// TIA Portal project "项目1" (V16)

(* hardware
DEVICE "HMI_1"  TP1200 Comfort
   slot 0: "HMI_1"  TP1200 Comfort  6AV2 124-0MC01-0AX0  16.0.0.0
   slot 1: "HMI_RT_1"  TP1200 Comfort  6AV2 124-0MC01-0AX0  16.0.0.0
   slot 5: "HMI_1.IE_CP_1"  PROFINET Interface  16.0.0.0
      slot 1: "PROFINET Interface_1"  PROFINET Interface
         slot 1: "Port_1"  Port
         slot 2: "Port_2"  Port
   slot 7: "HMI_1.MPI/DP_CP_1"  MPI/DP Interface  16.0.0.0
DEVICE "S7-1200 station_1"  S7-1200 Station
   slot 0: "Rack_0"  S7-1200 Rack  Rack  V1.0
   slot 1: "PLC_1"  CPU 1214C DC/DC/DC  6ES7 214-1AG40-0XB0  V4.4
*)

// ===== PLC "PLC_1"  CPU 1214C DC/DC/DC =====

VAR_GLOBAL   // PLC tag table "默认变量表"
   "正向" AT %M2.0 : Bool;
   "正向转动" AT %Q0.0 : Bool;
   "反向" AT %M2.1 : Bool;
   "停止" AT %M2.2 : Bool;
   "反向转动" AT %Q0.1 : Bool;
   "Clock_Byte" AT %MB100 : Byte;
   "Clock_10Hz" AT %M100.0 : Bool;
   "Clock_5Hz" AT %M100.1 : Bool;
   "Clock_2Hz" AT %M100.3 : Bool;
   "Clock_1.25Hz" AT %M100.4 : Bool;
   "Clock_1Hz" AT %M100.5 : Bool;   // 已用
   "Clock_0.625Hz" AT %M100.6 : Bool;
   "Clock_0.5Hz" AT %M100.7 : Bool;   // 已用
   "tag1" AT %M0.0 : Bool;
   "tag2" AT %M0.1 : Bool;
   "tag3" AT %M100.2 : Bool;   // 已用
   "tag4" AT %MW10 : Word;
   "tag6" AT %M1.3 : Bool;
   "低水位" AT %M3.0 : Bool;
   "高水位" AT %M3.2 : Bool;
   "供水泵" AT %M3.3 : Bool;
   "抽水" AT %M3.4 : Bool;
   "抽水泵" AT %M3.5 : Bool;
   "箭头动画2" AT %M4.1 : Bool;
   "箭头动画1" AT %M4.0 : Bool;
   "箭头动画3" AT %M4.3 : Bool;
   "箭头动画4" AT %MW11 : Int;
   "除污机工作" AT %M1.2 : Bool;
   "二箭头动画" AT %MW12 : Int;
   "二箭头动画2" AT %M4.5 : Bool;
   "二箭头动画3" AT %M4.6 : Bool;
   "密封池高水位" AT %M5.0 : Bool;
   "密封池低水位" AT %M5.1 : Bool;
   "密封池供水" AT %M5.2 : Bool;
   "空压机工作" AT %M5.3 : Bool;
   "滗水器工作" AT %M5.4 : Bool;
   "沉淀池供水" AT %M5.5 : Bool;
   "沉淀池高水位" AT %M5.6 : Bool;
   "沉淀池低水位" AT %M5.7 : Bool;
END_VAR

FUNCTION "块_1" : Void   // FC1, LAD
{ S7_Optimized_Access := 'TRUE' }
VERSION : 0.1
BEGIN
END_FUNCTION

ORGANIZATION_BLOCK "Main"   // OB1, LAD, ProgramCycle
TITLE = "Main Program Sweep (Cycle)"
{ S7_Optimized_Access := 'TRUE' }
VERSION : 0.1
   VAR_INPUT
      Initial_Call : Bool;   // Initial call of this OB
      Remanence : Bool;   // =True, if remanent data are available
   END_VAR
   VAR_TEMP   // added for the SCL form of the ladder/FBD networks
      _w1 : Bool;
   END_VAR
BEGIN

REGION Network 1
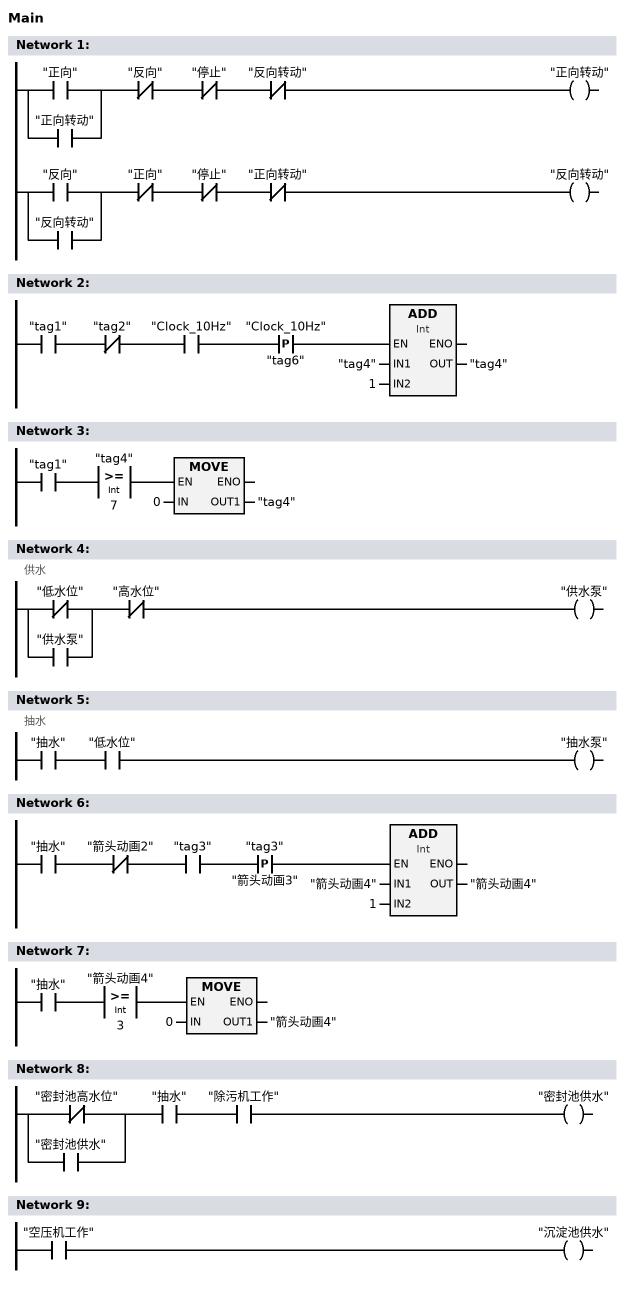
   RUNG wire#powerrail
      Contact( "正向" )
      wire#w1
      I_Contact( "反向" )
      I_Contact( "停止" )
      I_Contact( "反向转动" )
      Coil( "正向转动" )
   END_RUNG
   RUNG wire#powerrail
      Contact( "正向转动" )
   END_RUNG wire#w1
   RUNG wire#powerrail
      Contact( "反向" )
      wire#w2
      I_Contact( "正向" )
      I_Contact( "停止" )
      I_Contact( "正向转动" )
      Coil( "反向转动" )
   END_RUNG
   RUNG wire#powerrail
      Contact( "反向转动" )
   END_RUNG wire#w2
   // the same network as SCL:
   "正向转动" := ("正向" OR "正向转动") AND NOT "反向" AND NOT "停止" AND NOT "反向转动";
   "反向转动" := ("反向" OR "反向转动") AND NOT "正向" AND NOT "停止" AND NOT "正向转动";
END_REGION

REGION Network 2
   RUNG wire#powerrail
      Contact( "tag1" )
      I_Contact( "tag2" )
      Contact( "Clock_10Hz" )
      P_Contact(operand := "Clock_10Hz", bit := "tag6")
      { S7_Templates := "SrcType := Int" } Add(in1 := "tag4", in2 := 1, out => "tag4")
   END_RUNG
   // the same network as SCL:
   #_w1 := "tag1" AND NOT "tag2" AND "Clock_10Hz" AND "Clock_10Hz" AND NOT "tag6";   // rising edge of "Clock_10Hz"
   "tag6" := "Clock_10Hz";
   IF #_w1 THEN "tag4" := "tag4" + 1; END_IF;
END_REGION

REGION Network 3
   RUNG wire#powerrail
      Contact( "tag1" )
      { S7_Templates := "SrcType := Int" } GE_Contact(in1 := "tag4", in2 := 7)
      Move(in := 0, out1 => "tag4")
   END_RUNG
   // the same network as SCL:
   IF "tag1" AND ("tag4" >= 7) THEN "tag4" := 0; END_IF;
END_REGION

REGION Network 4
   // 供水
   RUNG wire#powerrail
      I_Contact( "低水位" )
      wire#w1
      I_Contact( "高水位" )
      Coil( "供水泵" )
   END_RUNG
   RUNG wire#powerrail
      Contact( "供水泵" )
   END_RUNG wire#w1
   // the same network as SCL:
   "供水泵" := (NOT "低水位" OR "供水泵") AND NOT "高水位";
END_REGION

REGION Network 5
   // 抽水
   RUNG wire#powerrail
      Contact( "抽水" )
      Contact( "低水位" )
      Coil( "抽水泵" )
   END_RUNG
   // the same network as SCL:
   "抽水泵" := "抽水" AND "低水位";
END_REGION

REGION Network 6
   RUNG wire#powerrail
      Contact( "抽水" )
      I_Contact( "箭头动画2" )
      Contact( "tag3" )
      P_Contact(operand := "tag3", bit := "箭头动画3")
      { S7_Templates := "SrcType := Int" } Add(in1 := "箭头动画4", in2 := 1, out => "箭头动画4")
   END_RUNG
   // the same network as SCL:
   #_w1 := "抽水" AND NOT "箭头动画2" AND "tag3" AND "tag3" AND NOT "箭头动画3";   // rising edge of "tag3"
   "箭头动画3" := "tag3";
   IF #_w1 THEN "箭头动画4" := "箭头动画4" + 1; END_IF;
END_REGION

REGION Network 7
   RUNG wire#powerrail
      Contact( "抽水" )
      { S7_Templates := "SrcType := Int" } GE_Contact(in1 := "箭头动画4", in2 := 3)
      Move(in := 0, out1 => "箭头动画4")
   END_RUNG
   // the same network as SCL:
   IF "抽水" AND ("箭头动画4" >= 3) THEN "箭头动画4" := 0; END_IF;
END_REGION

REGION Network 8
   RUNG wire#powerrail
      I_Contact( "密封池高水位" )
      wire#w1
      Contact( "抽水" )
      Contact( "除污机工作" )
      Coil( "密封池供水" )
   END_RUNG
   RUNG wire#powerrail
      Contact( "密封池供水" )
   END_RUNG wire#w1
   // the same network as SCL:
   "密封池供水" := (NOT "密封池高水位" OR "密封池供水") AND "抽水" AND "除污机工作";
END_REGION

REGION Network 9
   RUNG wire#powerrail
      Contact( "空压机工作" )
      Coil( "沉淀池供水" )
   END_RUNG
   // the same network as SCL:
   "沉淀池供水" := "空压机工作";
END_REGION
END_ORGANIZATION_BLOCK

(* ===== HMI "HMI_RT_1" =====
system functions are stored by id; their names below are inferred from use
connection "HMI_连接_2": ETHERNET, S7_1200_OMS

HMI tags "默认变量表"
   "Tag_ScreenNumber" : UInt AT %DB1.DBW0
   "正向" : Bool = PLC 正向 AT %M2.0, 1 s
   "反向" : Bool = PLC 反向 AT %M2.1, 1 s
   "停止" : Bool = PLC 停止 AT %M2.2, 1 s
   "反向转动" : Bool = PLC 反向转动 AT %Q0.1, 1 s
   "正向转动" : Bool = PLC 正向转动 AT %Q0.0, 1 s
   "P_N" : Bool = PLC tag2 AT %M0.1, 1 s
   "SPEED" : Word = PLC tag4 AT %MW10, 100 ms
   "toggle" : Bool = PLC tag1 AT %M0.0, 1 s

HMI tags "变量表_1"
   "高水位" : Bool = PLC 高水位 AT %M3.2, 100 ms
   "低水位" : Bool = PLC 低水位 AT %M3.0, 100 ms
   "供水泵" : Bool = PLC 供水泵 AT %M3.3, 100 ms
   "抽水" : Bool = PLC 抽水 AT %M3.4, 100 ms
   "抽水泵" : Bool = PLC 抽水泵 AT %M3.5, 100 ms
   "液位" : Int AT %DB1.DBW0
   "Clock_1Hz" : Bool = PLC Clock_1Hz AT %M100.5, 500 ms
      on ChangeValue: "VBFunction_1"(); "VBFunction_2"(); "VBFunction_3"()
   "箭头动画4" : Int = PLC 箭头动画4 AT %MW11, 100 ms
   "除污机工作" : Bool = PLC 除污机工作 AT %M1.2, 100 ms
   "二箭头动画" : Int = PLC 二箭头动画 AT %MW12, 100 ms
   "密封池高水位" : Bool = PLC 密封池高水位 AT %M5.0, 100 ms
   "密封池低水位" : Bool = PLC 密封池低水位 AT %M5.1, 100 ms
   "密封池供水" : Bool = PLC 密封池供水 AT %M5.2, 100 ms
   "空压机工作" : Bool = PLC 空压机工作 AT %M5.3, 100 ms
   "密封池液位" : Int AT %DB1.DBX0.0
   "滗水器工作" : Bool = PLC 滗水器工作 AT %M5.4, 100 ms
   "沉淀池供水" : Bool = PLC 沉淀池供水 AT %M5.5, 100 ms
   "沉淀池液位" : Int AT %DB1.DBX0.0
   "沉淀池高水位" : Bool = PLC 沉淀池高水位 AT %M5.6, 100 ms
   "沉淀池低水位" : Bool = PLC 沉淀池低水位 AT %M5.7, 100 ms

graphic list "rotation": 0 '风扇1'; 1 '风扇2_1'; 2 '风扇3_1'; 3 '风扇4'; 4 '风扇5'; 5 '风扇6'; 6 '风扇7'

graphic list "arrows_1": 0 '箭头2_0'; 1 '箭头2_4'; 2 '箭头2_3'

graphic list "arrows_2": 0 '竖向箭头1_0'; 1 '竖向箭头1_1'; 2 '竖向箭头1_2'

graphic list "arrows_3": 0 '箭头2_5'; 1 '反方向箭头1'; 2 '反方向箭头2'

screen "根画面" 1280x733, template "模板_1"
   on GenerateScreen: SetTag("Tag_ScreenNumber", 1)
   TextField "HmiScreenItemData" at 52,22 size 1024x27; Text '你好 / 欢迎进入 HMI_1 (TP1200 Comfort)！'
   Button "按钮_1" at 104,159 size 157x55; TextOff '电机正转'
      on Press: SetBit("正向")
      on Release: ResetBit("正向")
   Button "按钮_2" at 103,243 size 157x55; TextOff '电机反转'
      on Press: SetBit("反向")
      on Release: ResetBit("反向")
   Button "按钮_3" at 104,325 size 157x55; TextOff '停止'
      on Press: SetBit("停止")
      on Release: ResetBit("停止")
   Circle "圆_1" at 298,174 size 42x42
      Appearance <- "正向转动"
   Circle "圆_2" at 298,257 size 42x42
      Appearance <- "反向转动"

Template "模板_1" 1280x733
   Button "Exit" at 1200,679 size 78x59; TextOff 'Exit / 退出'; PictureOff "ExitRuntime_TP1200_Comfort_TR"; PictureOn "ExitRuntime_TP1200_Comfort_TR"
      on Release: StopRuntime(0)
   Button "Language" at 1120,679 size 78x59; TextOff 'Language / 语言'; PictureOff "ToggleLanguage_TP1200_Comfort_TR"; PictureOn "ToggleLanguage_TP1200_Comfort_TR"
      on Release: function_fb9197e8(-1)
   Button "Template_Button" at 1040,679 size 78x59; TextOff 'Text'
   Button "Template_Button_1" at 960,679 size 78x59; TextOff 'Text'
   Button "Template_Button_2" at 880,679 size 78x59; TextOff 'Text'
   Button "Template_Button_3" at 800,679 size 78x59; TextOff 'Text'
   Button "Template_Button_4" at 720,679 size 78x59; TextOff 'Text'
   Button "Template_Button_5" at 640,679 size 78x59; TextOff 'Text'
   Button "Template_Button_6" at 561,679 size 78x59; TextOff 'Text'
   Button "Template_Button_7" at 481,679 size 78x59; TextOff 'Text'
   Button "Template_Button_8" at 401,679 size 78x59; TextOff 'Text'
   Button "Template_Button_9" at 321,679 size 78x59; TextOff 'Text'
   Button "Template_Button_10" at 241,679 size 78x59; TextOff 'Text'
   Button "Template_Button_11" at 161,679 size 78x59; TextOff 'Text'
   Button "Alarms" at 81,679 size 78x59; TextOff 'Alarms / 报警'; PictureOff "AlarmDisplay_TP1200_Comfort_TR"; PictureOn "AlarmDisplay_TP1200_Comfort_TR"
      on Release: function_ef3f5d25("报警窗口_Unacknowledged", -1)
   Button "Start screen" at 1,679 size 78x59; TextOff 'Start screen / 起始画面'; PictureOff "NavigateHome_TP1200_Comfort_TR"; PictureOn "NavigateHome_TP1200_Comfort_TR"
      on Release: ActivateScreen("根画面", 0)

screen "画面_1" 1280x733
   Group "Group_6" at 6,455 size 253x79; Picture "管道"
   Group "Group_7" at 118,405 size 310x305; Picture "污泥泵"
   Group "Group_8" at 285,336 size 342x197; Picture "滗水器"
   GraphicView "图形视图_15" at 590,381 size 226x261; Picture "蓄水罐"
   Group "Group_1" at 6,64 size 876x296; Picture "水泵"
   Group "Group_2" at 781,290 size 360x193; Picture "管道"
   Group "Group_3" at 2,24 size 154x61; Picture "管道"
   TextField "文本域_1" at 54,333 size 125x53; Text '储水罐'
   TextField "文本域_3" at 647,619 size 104x45; Text '密封池'
   TextField "文本域_4" at 393,660 size 74x33; Text '储泥罐'
   TextField "文本域_7" at 515,112 size 166x45; Text '一级除污机'
   TextField "文本域_8" at 713,132 size 166x45; Text '二级除污机'
   TextField "文本域_9" at 773,268 size 116x33; Text '液压感应器'
   TextField "文本域_5" at 581,366 size 74x33; Text '空压机'
   TextField "文本域_10" at 105,537 size 74x33; Text '污泥泵'
   TextField "文本域_11" at 781,369 size 116x33; Text '液位传感器'
   TextField "文本域_12" at 514,413 size 74x33; Text '滗水器'
   TextField "文本域_13" at 306,178 size 104x45; Text '抽水泵'
   TextField "文本域_14" at 9,8 size 104x45; Text '进水口'
   TextField "文本域_17" at 76,435 size 135x45; Text '出水管道'
   TextField "文本域_15" at 851,494 size 119x40; Text '系统设备'
   TextField "文本域_16" at 1101,494 size 119x40; Text '工作状态'
   Circle "圆_1" at 1148,541 size 26x26
      Appearance <- "供水泵"
   TextField "文本域_18" at 875,537 size 74x33; Text '进水口'
   TextField "文本域_19" at 875,576 size 74x33; Text '抽水泵'
   TextField "文本域_20" at 875,616 size 74x33; Text '空压机'
   TextField "文本域_21" at 875,656 size 74x33; Text '鼓风机'
   TextField "文本域_22" at 875,693 size 74x33; Text '滗水器'
   Circle "圆_2" at 1148,579 size 26x26
      Appearance <- "抽水泵"
   Circle "圆_3" at 1148,619 size 26x26
      Appearance <- "沉淀池供水"
   Circle "圆_4" at 1149,661 size 26x26
      Appearance <- "toggle"
   Circle "圆_5" at 1149,699 size 26x26
      Appearance <- "空压机工作"
   TextField "文本域_6" at 273,605 size 104x45; Text '沉淀池'
   TextField "文本域_2" at 1046,6 size 92x40; Text '控制台'
   Bar "棒图_1" at 33,118 size 182x210; MinimumValue 0; MaximumValue 100
      ProcessValue <- "液位"
   Group "Group_10" at 467,516 size 160x211; Picture "污泥泵"
   Rectangle "矩形_4" at 34,157 size 135x9
      Appearance <- "高水位"
   Rectangle "矩形_5" at 33,308 size 136x9
      Appearance <- "低水位"
   GraphicIOField "图形 I/O 域_3" at 227,261 size 62x29; PictureList "arrows_1"
      ProcessValue <- "箭头动画4"
      Visibility <- "抽水"
   GraphicIOField "图形 I/O 域_4" at 400,227 size 67x35; PictureList "arrows_1"
      ProcessValue <- "箭头动画4"
      Visibility <- "抽水"
   GraphicIOField "图形 I/O 域_5" at 469,225 size 67x36; PictureList "arrows_1"
      ProcessValue <- "箭头动画4"
      Visibility <- "抽水"
   Circle "圆_6" at 568,290 size 13x13
      Appearance <- "除污机工作"
   Circle "圆_7" at 747,317 size 13x13
      Appearance <- "除污机工作"
   GraphicIOField "图形 I/O 域_6" at 924,276 size 67x35; PictureList "arrows_1"
      Visibility <- "除污机工作"
      ProcessValue <- "箭头动画4"
   GraphicIOField "图形 I/O 域_7" at 1008,276 size 67x35; PictureList "arrows_1"
      Visibility <- "除污机工作"
      ProcessValue <- "箭头动画4"
   GraphicIOField "图形 I/O 域_8" at 1125,348 size 36x65; PictureList "arrows_2"
      ProcessValue <- "箭头动画4"
      Visibility <- "除污机工作"
   GraphicIOField "图形 I/O 域_2" at 969,408 size 77x38; PictureList "arrows_3"
      Visibility <- "除污机工作"
      ProcessValue <- "箭头动画4"
   GraphicIOField "图形 I/O 域_9" at 880,408 size 77x38; PictureList "arrows_3"
      ProcessValue <- "箭头动画4"
      Visibility <- "除污机工作"
   Button "按钮_1" at 949,53 size 96x32; TextOff '抽水泵'
      on Click: InvertBit("抽水"); ResetBit("toggle")
   Button "按钮_2" at 949,147 size 96x32; TextOff '鼓风机'
      on Click: InvertBit("toggle"); ResetBit("抽水"); ResetBit("除污机工作")
   Bar "棒图_2" at 613,430 size 167x188; MinimumValue 0; MaximumValue 100
      ProcessValue <- "密封池液位"
   Button "按钮_3" at 949,100 size 96x32; TextOff '除污机'
      on Click: InvertBit("除污机工作"); ResetBit("toggle")
   GraphicIOField "图形 I/O 域_1" at 700,433 size 52x51; PictureList "rotation"
      ProcessValue <- "SPEED"
   TextField "文本域_23" at 693,399 size 74x33; Text '鼓风机'
   Group "Group_4" at 642,349 size 65x107; Picture "空压机"
   Circle "圆_8" at 676,376 size 10x10
      Appearance <- "沉淀池供水"
   Circle "圆_9" at 738,433 size 10x10
      Appearance <- "toggle"
   Button "按钮_4" at 949,191 size 96x32; TextOff '空压机'
      on Click: InvertBit("空压机工作"); InvertBit("滗水器工作"); ResetBit("抽水"); ResetBit("除污机工作"); ResetBit("toggle")
   Circle "圆_10" at 547,494 size 10x10
      Appearance <- "沉淀池供水"
   Rectangle "矩形_6" at 616,471 size 80x9
      Appearance <- "密封池高水位"
   Rectangle "矩形_7" at 616,597 size 80x9
      Appearance <- "密封池低水位"
   Group "Group_9" at 752,366 size 38x168; Picture "液位传感器"
   Bar "棒图_3" at 257,446 size 141x164; MinimumValue 0; MaximumValue 100
      ProcessValue <- "沉淀池液位"
   Rectangle "矩形_8" at 259,471 size 80x9
      Appearance <- "沉淀池高水位"
   Rectangle "矩形_9" at 259,592 size 80x9
      Appearance <- "密封池低水位"
   Group "Group_11" at 639,53 size 120x25
   GraphicView "图形视图_3" at 264,207 size 162x153; Picture "水泵"
   GraphicView "图形视图_2" at 216,294 size 80x31; Picture "管道"
   GraphicView "图形视图_1" at 6,64 size 249x292; Picture "蓄水罐"
   Group "Group" at 6,64 size 420x296; Picture "水泵"
   GraphicView "图形视图_4" at 401,244 size 143x58; Picture "管道"
   GraphicView "图形视图_5" at 539,159 size 141x164; Picture "除污机"
   GraphicView "图形视图_6" at 677,264 size 41x69; Picture "管道"
   GraphicView "图形视图_7" at 710,177 size 172x176; Picture "除污机"
   GraphicView "图形视图_8" at 879,290 size 96x65; Picture "管道"
   GraphicView "图形视图_9" at 972,291 size 96x65; Picture "管道"
   GraphicView "图形视图_10" at 1062,305 size 59x52; Picture "弯曲管道"
   GraphicView "图形视图_11" at 1062,354 size 79x72; Picture "管道2"
   GraphicView "图形视图_12" at 1066,415 size 59x52; Picture "弯曲管道2"
   GraphicView "图形视图_13" at 869,424 size 199x59; Picture "管道"
   GraphicView "图形视图_14" at 781,389 size 90x93; Picture "管道节点"
   GraphicView "图形视图_16" at 642,349 size 65x39; Picture "空压机"
   GraphicView "图形视图_17" at 644,388 size 59x68; Picture "管道2"
   GraphicView "图形视图_19" at 534,516 size 93x115; Picture "污泥泵"
   GraphicView "图形视图_20" at 509,589 size 41x39; Picture "弯曲管道3"
   GraphicView "图形视图_18" at 467,620 size 91x107; Picture "储泥罐_1"
   GraphicView "图形视图_21" at 501,434 size 116x99; Picture "滗水器"
   Group "Group_5" at 285,336 size 342x111; Picture "管道2"
   GraphicView "图形视图_23" at 567,386 size 60x61; Picture "管道2"
   GraphicView "图形视图_24" at 568,345 size 43x41; Picture "弯曲管道"
   GraphicView "图形视图_22" at 340,336 size 233x48; Picture "管道"
   GraphicView "图形视图_25" at 298,344 size 46x44; Picture "弯曲管道3"
   GraphicView "图形视图_26" at 285,386 size 54x46; Picture "管道2"
   GraphicView "图形视图_28" at 174,509 size 97x99; Picture "污泥泵"
   GraphicView "图形视图_29" at 152,571 size 40x36; Picture "弯曲管道3"
   GraphicView "图形视图_30" at 118,604 size 93x106; Picture "储泥罐_1"
   GraphicView "图形视图_27" at 235,405 size 193x222; Picture "蓄水罐"
   GraphicView "图形视图_31" at 174,480 size 85x53; Picture "管道"
   GraphicView "图形视图_32" at 96,455 size 83x75; Picture "管道节点"
   GraphicView "图形视图_33" at 6,480 size 92x54; Picture "管道"
   GraphicView "图形视图_34" at 2,24 size 106x60; Picture "管道"
   GraphicView "图形视图_35" at 106,37 size 50x48; Picture "弯曲管道"
   GraphicView "图形视图_36" at 752,366 size 38x67; Picture "液位传感器"
   IOField "I/O 域_2" at 639,65 size 5x0; FormatPattern 1
      ProcessValue <- "Clock_1Hz"
   TextField "文本域_24" at 668,53 size 91x25; Text 'by 侯翰亭'

VB script "VBFunction_1"
   '提示：
   ' 1. 使用 <CTRL+SPACE> 或 <CTRL+I> 快捷键打开含所有对象和函数的列表
   ' 2. 使用 HMI Runtime 对象写入代码。
   '  示例：HmiRuntime.Screens("Screen_1")。
   ' 3. 使用 <CTRL+J> 快捷键创建对象引用。
   '从此位置起写入代码：
   Dim startAdd,startsub,LevelData,HighLevel,LowLevel
   
   Set startAdd=SmartTags("供水泵")
   Set startsub=SmartTags("抽水泵")
   'write
   Set LevelData=SmartTags("液位")
   Set HighLevel=SmartTags("高水位")
   Set LowLevel=SmartTags("低水位")
   
   If startAdd=True And LevelData<80 Then
   	LevelData.Value=LevelData.Value+4
   End If
   
   '液位下降
   If startsub=True And LevelData>=5 Then
   	LevelData.Value=LevelData.Value-5
   End If
   
   '到达高料位
   If LevelData.Value>=80 Then
   	HighLevel.Value=True
   Else
   	HighLevel.Value=False
   End If
   '到达低料位
   If LevelData.Value>=5 Then
   	LowLevel.Value=True
   Else
   	LowLevel.Value=False
   
   End If

VB script "VBFunction_2"
   '提示：
   ' 1. 使用 <CTRL+SPACE> 或 <CTRL+I> 快捷键打开含所有对象和函数的列表
   ' 2. 使用 HMI Runtime 对象写入代码。
   '  示例：HmiRuntime.Screens("Screen_1")。
   ' 3. 使用 <CTRL+J> 快捷键创建对象引用。
   '从此位置起写入代码：
   Dim Add1,Add2,suck,waterLevel,High,Low,bibi
   
   Set Add1=SmartTags("抽水")
   Set Add2=SmartTags("除污机工作")
   
   Set suck=SmartTags("空压机工作")
   Set bibi=SmartTags("沉淀池供水")
   'write
   Set waterLevel=SmartTags("密封池液位")
   Set High=SmartTags("密封池高水位")
   Set Low=SmartTags("密封池低水位")
   
   If Add1.Value=True And Add1.Value=True And waterLevel.Value>=80 Then
   	Add1.Value=False
   	Add2.Value=False
   End If
   
   If waterLevel.Value<=10 Then
   	suck.Value=False
   	bibi.Value=False
   End If
   
   If Add1.Value=True And Add2.Value=True And waterLevel.Value<80 Then
   	waterLevel.Value=waterLevel.Value+2
   End If
   
   '液位下降
   If suck=True And waterLevel>=10 Then
   	waterLevel.Value=waterLevel.Value-3
   End If
   
   '到达高料位
   If waterLevel.Value>=80 Then
   	High.Value=True
   Else
   	High.Value=False
   End If
   
   '到达低料位
   If waterLevel.Value>=10 Then
   	Low.Value=True
   Else
   	Low.Value=False
   
   End If

VB script "VBFunction_3"
   '提示：
   ' 1. 使用 <CTRL+SPACE> 或 <CTRL+I> 快捷键打开含所有对象和函数的列表
   ' 2. 使用 HMI Runtime 对象写入代码。
   '  示例：HmiRuntime.Screens("Screen_1")。
   ' 3. 使用 <CTRL+J> 快捷键创建对象引用。
   '从此位置起写入代码：
   
   Dim suck1,Level2,HighL,LowL
   
   Set suck1=SmartTags("沉淀池供水")
   'write
   Set Level2=SmartTags("沉淀池液位")
   Set HighL=SmartTags("沉淀池高水位")
   Set LowL=SmartTags("沉淀池低水位")
   
   If suck1.Value=True And Level2.Value>=80 Then
   	suck1.Value=False
   End If
   
   If suck1.Value=True And Level2.Value<80 Then
   	Level2.Value=Level2.Value+2
   End If
   
   '液位下降
   If Level2>=10 Then
   	Level2.Value=Level2.Value-1
   End If
   
   '到达高料位
   If Level2.Value>=80 Then
   	HighL.Value=True
   Else
   	HighL.Value=False
   End If
   
   '到达低料位
   If Level2.Value>=10 Then
   	LowL.Value=True
   Else
   	LowL.Value=False
   End If
*)